// TwinCAT 3 PLC project Untitled1
// ProgramVersion: 3.1.4024.0
// libraries:
//   Tc2_Standard, * (Beckhoff Automation GmbH)
//   Tc2_System, * (Beckhoff Automation GmbH)
//   Tc3_Module, * (Beckhoff Automation GmbH)
// project tree:
//   FB/ FB_ST10.TcPOU
//   / PlcTask.TcTTO
//   POUs/ MAIN.TcPOU
// real-time tasks:
//   TASK PlcTask: cycle T#10ms, priority 20, ADS port 350

CONFIGURATION Untitled1
    RESOURCE PLC ON TwinCAT3
        TASK PlcTask(INTERVAL := T#10ms, PRIORITY := 20);
        PROGRAM MAIN WITH PlcTask : MAIN;
    END_RESOURCE
END_CONFIGURATION

// ---- POUs/MAIN.TcPOU
PROGRAM MAIN
VAR
END_VAR

END_PROGRAM

// ---- FB/FB_ST10.TcPOU
FUNCTION_BLOCK FB_ST10
VAR
	_Camera : BOOL;
	_Scanner : BOOL;
	_triger : BOOL;
	_busy  : BOOL;
	_desc : STRING;
END_VAR

METHOD PROTECTED _camera
VAR_INPUT
END_VAR
IF _Camera THEN 
	_desc:= 'Camera ready';
ELSIF _triger THEN 
	_desc:= 'Triger';
ELSE
	_busy:= FALSE;
END_IF
END_METHOD

END_FUNCTION_BLOCK
